TYPE "Prod_SetUp_Man_Feedbak"
VERSION : 0.1
// Block: Prod_SetUp_Man_Feedbak
   STRUCT
      Done : Bool;
      Done_X : Bool;
      Done_Y : Bool;
      Done_Z : Bool;
      Ack_Eseguito_X : Array[1..SETUP_MAN_OPERATIONS_QTY] of Bool;
      Ack_Eseguito_Y : Array[1..SETUP_MAN_OP_WITH_CODE_QTY] of Bool;
   END_STRUCT;

END_TYPE
